// TIA Portal V17 export
// export: Created 2024-08-07T21:44:16.4334782Z, ExportSetting WithDefaults, DisplayName Totally Integrated Automation Portal, DisplayVersion V17 Update 7, DisplayName TIA Portal Openness, DisplayVersion V17 Update 7, DisplayName TIA Portal Version Control Interface, DisplayVersion V17, DisplayName SINAMICS Startdrive Advanced, DisplayVersion V17 SP2, DisplayName SINAMICS Startdrive G110M, G120, G120C, G120D, G120P, G115D, DisplayVersion V17 SP2, DisplayName SINAMICS Startdrive G130, G150, S120, S150, SINAMICS MV, S210, DisplayVersion V17 SP2, DisplayName STEP 7 Professional, DisplayVersion V17 Update 7, DisplayName STEP 7 Safety, DisplayVersion V17 Update 6, DisplayName WinCC Advanced / Unified PC, DisplayVersion V17 Update 7
TYPE "connectionParameterType"
// stored: IsFailsafeCompliant false
   STRUCT
      ConnectInfo { ExternalAccessible := 'False'; ExternalVisible := 'False'; ExternalWritable := 'False'; S7_SetPoint := 'True'} : OPC_UA_SessionConnectInfo;
      ConnectionHdl { ExternalAccessible := 'False'; ExternalVisible := 'False'; ExternalWritable := 'False'} : DWord;
      ServerEndpointUrl { ExternalAccessible := 'False'; ExternalVisible := 'False'; ExternalWritable := 'False'} : String[254] := 'opc.tcp://192.168.0.2:4840';
   END_STRUCT;
   // ConnectInfo.SessionName := WSTRING#'OPC UA Connection_1';
   // ConnectInfo.ApplicationName := WSTRING#'';
   // ConnectInfo.SecurityMsgMode := 1;
   // ConnectInfo.SecurityPolicy := 1;
   // ConnectInfo.ServerUri := '';
   // ConnectInfo.CheckServerCertificate := False;
   // ConnectInfo.TransportProfile := 1;
   // ConnectInfo.UserIdentityTokenType := 0;
   // ConnectInfo.CertificateID := 0;
   // ConnectInfo.SessionTimeout := T#30S;
   // ConnectInfo.MonitorConnection := T#5S;
   // ConnectInfo.LocaleIDs[0] := 'en-US';
   // ConnectInfo.LocaleIDs[1..4] := '';
END_TYPE
